// SIMATIC S7-200 project (STEP 7-Micro/WIN), CPU 226 CN REL 02.01

ORGANIZATION_BLOCK 主程序:OB1
TITLE=
BEGIN
Network 2
//  初始化高速计数器与定时中断 (仅首次上电执行一次)
LD     SM0.1
MOVB   16#F8, SMB37
HDEF   0, 9
MOVD   0, SMD38
HSC    0
MOVB   50, SMB34             // 50ms 中断采样率
ATCH   INT_0:INT0, 10
ENI
MOVW   0, VW100              // 状态机初始为 0
// === 双闭环核心参数初始化 ===
MOVR   0.0, VD130            // 上次位置初值清零 (用于测速)
MOVR   0.0, VD154            // 速度环积分器清零
// 1. 位置外环比例 Kp_pos (控制减速距离)
// 建议值小一点，比如 0.5。误差1000个脉冲时，要求速度为 500脉冲/50ms
MOVR   0.5, VD120
// 2. 速度内环比例 Kp_spd (控制爆发力)
// 建议值：10.0。速度每差 1个脉冲/50ms，补 10 对应电压
MOVR   10.0, VD146
// 3. 速度内环积分 Ki_spd (消除稳态静差，爬进终点全靠它)
// 建议值：0.5。
MOVR   0.5, VD150
Network 3
//  外部启动开关 (I0.2)，触发折返跑任务
LD     I0.2
EU                           // 上升沿触发
MOVB   16#C8, SMB37          // 指令：仅更新当前值
MOVD   0, SMD38              // 无论当前在哪，强制将脉冲清零作为绝对起点
HSC    0
MOVW   1, VW100              // 切换到 状态1：准备第一段正向冲刺


Network 4
//  状态 1：正向 3 圈 (目标设为 +1200 脉冲)
Network 5
//  状态 1：正向 3 圈 (目标设为 +1200 脉冲)
LDW=   VW100, 1
MOVR   1200.0, VD104


LDW=   VW100, 1              // 【核心修复】：必须前提是处于状态 1
AD>=   HC0, 1190             // 且脉冲跑到 1190 以上
A      M0.0                  // 且 PID 确认到位
S      M1.1, 1


LD     M1.1
TON    T37, 5                // 稳住 0.5 秒


LD     T37
R      M1.1, 1
R      M0.0, 1
MOVW   2, VW100              // 切换到 状态2
Network 6
//  状态 2：反向 3 圈 (目标设为回到 0 脉冲处)
Network 7
//  状态 2：反向 3 圈 (目标设为回到 0 脉冲处)
LDW=   VW100, 2
MOVR   0.0, VD104


LDW=   VW100, 2              // 【核心修复】：必须前提是处于状态 2
AD<=   HC0, 10               // 且脉冲退回 10 以内
A      M0.0
S      M1.2, 1


LD     M1.2
TON    T38, 5                // 稳住 0.5 秒


LD     T38
R      M1.2, 1
R      M0.0, 1
MOVW   3, VW100              // 切换到 状态3
Network 8
//  状态 3：最后一次正向 3 圈 (目标再次设为 +1200 脉冲)
Network 9
//  状态 3：最后一次正向 3 圈 (目标再次设为 +1200 脉冲)
LDW=   VW100, 3
MOVR   1200.0, VD104


LDW=   VW100, 3              // 【核心修复】：必须前提是处于状态 3
AD>=   HC0, 1190
A      M0.0
S      M1.3, 1


LD     M1.3
TON    T39, 5                // 稳住 0.5 秒


LD     T39
R      M1.3, 1
R      M0.0, 1
MOVW   4, VW100              // 状态4：任务完美结束！
Network 11 // 网络标题
// 网络注释
END_ORGANIZATION_BLOCK

// SBR1: protected block, not included

INTERRUPT_BLOCK INT_0:INT0
TITLE=
BEGIN
Network 2
//  1. 读取当前位置，并测算实时速度
LD     SM0.0
MOVD   HC0, AC0
DTR    AC0, AC0
MOVR   AC0, VD108            // 记录当前位置 PV


MOVR   VD108, AC1
-R     VD130, AC1            // 当前位置 - 上次位置
MOVR   AC1, VD134            // = 【当前实时速度】 (脉冲数/50ms)
MOVR   VD108, VD130          // 将当前位置保存，供下周期使用


Network 3
//  2. 计算位置误差
LD     SM0.0
MOVR   VD104, AC0            // 目标位置 SP
-R     VD108, AC0
MOVR   AC0, VD112            // 【位置误差】 (带正负号)


Network 4
//  3. 纯数学求绝对位置误差 (用于死区判断)
LD     SM0.0
MOVR   VD112, VD116
LDR<   VD116, 0.0
*R     -1.0, VD116


Network 5
//  4. 到位死区判定，并清空积分器 (防积分饱和)
LDR<=  VD116, 5.0
=      M0.0                  // 触碰死区线，M0.0 置位
LD     M0.0
MOVR   0.0, VD154            // 只要进入死区，立刻清零速度环积分器！


Network 6
//  5. 【位置外环 P 控制】：计算出目标速度
LD     SM0.0
MOVR   VD112, AC0
*R     VD120, AC0            // 目标速度 = 位置误差 * 位置Kp


// 外环限幅
                     // 外环限幅
LDR>   AC0, 1500.0
MOVR   1500.0, AC0
LDR<   AC0, -1500.0
MOVR   -1500.0, AC0


LD     SM0.0                 // <--- 【Bug 修复 1：恢复堆栈！】
MOVR   AC0, VD138            // 更新目标速度


Network 7
//  6. 算出速度误差
LD     SM0.0
MOVR   VD138, AC0            // 目标速度
-R     VD134, AC0            // - 实时速度
MOVR   AC0, VD142            // = 【速度误差】


Network 8
//  7. 【速度内环 PI 控制】：算出最终电压输出
LD     SM0.0
// 算比例项 (P)
                 // 算比例项 (P)
MOVR   VD142, AC1
*R     VD146, AC1            // 速度误差 * 速度Kp


// 算积分项 (I)
                 // 算积分项 (I)
LD     SM0.0                 // <--- 【规范化堆栈】
MOVR   VD142, AC2
*R     VD150, AC2            // 速度误差 * 速度Ki
+R     VD154, AC2            // 累加上一次的积分值


// 积分限幅
                     // 积分限幅
LDR>   AC2, 32000.0
MOVR   32000.0, AC2
LDR<   AC2, -32000.0
MOVR   -32000.0, AC2


LD     SM0.0                 // <--- 【Bug 修复 2：恢复堆栈！】
MOVR   AC2, VD154            // 更新积分器


// P + I 合并
                 // P + I 合并
LD     SM0.0                 // <--- 【Bug 修复 3：恢复堆栈！】
+R     AC2, AC1              // 比例项 + 积分项
MOVR   AC1, VD158            // = 【PID 最终输出】


Network 9
//  8. 提取绝对电压值
LD     SM0.0
MOVR   VD158, VD124
LDR<   VD124, 0.0
*R     -1.0, VD124           // 取绝对值作为 0-10V 电压


LDR>   VD124, 32000.0
MOVR   32000.0, VD124        // 最高限幅 10V


Network 10
//  9. 动作分配：如果输出为正，正转
LDN    M0.0
AW<>   VW100, 0
AW<>   VW100, 4
AR>    VD158, 0.0            // 判断带符号的最终输出
S      Q0.0, 1
R      Q0.1, 1


Network 11
//  10. 动作分配：如果输出为负，反转
LDN    M0.0
AW<>   VW100, 0
AW<>   VW100, 4
AR<    VD158, 0.0
R      Q0.0, 1
S      Q0.1, 1


Network 12
//  11. 实时输出模拟量调速信号
LDN    M0.0
AW<>   VW100, 0
AW<>   VW100, 4
ROUND  VD124, AC0
DTI    AC0, VW200
MOVW   VW200, AQW0


Network 13
//  12. 终极刹车保护
LD     M0.0
OW=    VW100, 0
OW=    VW100, 4
R      Q0.0, 2
MOVW   0, AQW0
END_INTERRUPT_BLOCK

// (further data pages could not be read)
